// TwinCAT 3 PLC project my_plc
// ProgramVersion: 3.1.4026.20
// libraries:
//   Tc2_Standard, * (Beckhoff Automation GmbH)
//   Tc2_System, * (Beckhoff Automation GmbH)
// project tree:
//   / PlcTask.TcTTO
//   POUs/ FB_MyBlock.TcPOU, MAIN.TcPOU
// real-time tasks:
//   TASK PlcTask: cycle T#10ms, priority 20, ADS port 350

CONFIGURATION my_plc
    RESOURCE PLC ON TwinCAT3
        TASK PlcTask(INTERVAL := T#10ms, PRIORITY := 20);
        PROGRAM MAIN WITH PlcTask : MAIN;
    END_RESOURCE
END_CONFIGURATION

// ---- POUs/MAIN.TcPOU
PROGRAM MAIN
VAR
	fb		: FB_MyBlock();
END_VAR

fb();

END_PROGRAM

// ---- POUs/FB_MyBlock.TcPOU
FUNCTION_BLOCK FB_MyBlock
VAR_OUTPUT
	myVar		: INT := 42;
END_VAR

END_FUNCTION_BLOCK
